(* IEC 61131-3 sources: automatic-screwdriver-line/src/POU/Job_Handler, 6 files *)

(* ---- ErrorCodeToString.st ---- *)
// Generated from Automatic_ScrewDriver_Line.xml by tools/export_st.py - do not edit.
// The CODESYS project is the source of truth.

FUNCTION ErrorCodeToString : STRING
VAR_INPUT
	Code : ErrorCode;
END_VAR

CASE Code OF
	ErrorCode.NoError :
		ErrorCodeToString := 'No Error';
	ErrorCode.EnablementError:
		ErrorCodeToString := 'Enablement Error';
	ErrorCode.ScrewNotReleased:
		ErrorCodeToString := 'Screw Not Released';
	ErrorCode.TargetNotReached:
		ErrorCodeToString := 'Target Not Reached';
	ErrorCode.SpindleError:
		ErrorCodeToString := 'Spindle Error';
	ErrorCode.CobotNotConnected:
		ErrorCodeToString := 'Cobot Not Connected';
	ErrorCode.CobotMovementNotReached:
		ErrorCodeToString := 'Cobot Movement Not Reached';
	ErrorCode.RtcNotAvailable:
		ErrorCodeToString := 'Rtc Not Available';
ELSE
		ErrorCodeToString := 'Unknown Error';
END_CASE

END_FUNCTION

(* ---- Trace.st ---- *)
// Generated from Automatic_ScrewDriver_Line.xml by tools/export_st.py - do not edit.
// The CODESYS project is the source of truth.

FUNCTION Trace : BOOL
VAR_INPUT
	Severity : UDINT;   // LogClass.LOG_INFO / LOG_WARNING / LOG_ERROR
	Msg : STRING(255);
END_VAR

LogAdd(
	hLogger   := CmpLog.LogConstants.LOG_STD_LOGGER,
	stCmpName := Machine_Constants.LOG_COMPONENT_NAME,
	diClassID := UDINT_TO_DINT(Severity),
	diErrorID := 0,
	diInfoID  := 0,
	stInfo    := Msg
);

Trace := TRUE;

END_FUNCTION

(* ---- FB_JobManager.st ---- *)
// Generated from Automatic_ScrewDriver_Line.xml by tools/export_st.py - do not edit.
// The CODESYS project is the source of truth.

FUNCTION_BLOCK FB_JobManager EXTENDS FB_FunctionBlock_Base
VAR
	_InitDone : BOOL;
	_state : JobState;
	_ActiveError : ErrorCode;
	_Stop : BOOL;
	_Reseters : ARRAY[1..6] OF I_Resettable;
	_Diagnosable : ARRAY[1..6] OF I_Diagnosable;
	_i : DINT;
	_UserInterface : REFERENCE TO FB_UserInterface;
	_JobSelector : REFERENCE TO FB_JobSelector;
	_Mover : I_Mover;
	_zAxis : REFERENCE TO FB_zAxis;
	_Spindle : REFERENCE TO FB_Spindle;
	_ReportJob : REFERENCE TO FB_ReportJob;
	_SpindleOk : BOOL;
	_MoverOk : BOOL;
END_VAR

METHOD Reset : BOOL

ClearError();
Reset := TRUE;
END_METHOD

METHOD Init : BOOL
VAR_INPUT
	UserInterface : REFERENCE TO FB_UserInterface;
	JobSelector : REFERENCE TO FB_JobSelector;
	Mover : I_Mover;
	zAxis : REFERENCE TO FB_zAxis;
	Spindle : REFERENCE TO FB_Spindle;
	ReportJob : REFERENCE TO FB_ReportJob;
END_VAR

_UserInterface REF= UserInterface;
_JobSelector REF= JobSelector;
_Mover := Mover;
_zAxis REF= zAxis;
_Spindle REF= Spindle;
_ReportJob REF= ReportJob;

// Reseters
_Reseters[1] := _UserInterface;
_Reseters[2] := _JobSelector;
_Reseters[3] := _Mover;
_Reseters[4] := _zAxis;
_Reseters[5] := _Spindle;
_Reseters[6] := _ReportJob;

// Diagnosable
_Diagnosable[1] := _UserInterface;
_Diagnosable[2] := _JobSelector;
_Diagnosable[3] := _Mover;
_Diagnosable[4] := _zAxis;
_Diagnosable[5] := _Spindle;
_Diagnosable[6] := _ReportJob;

_InitDone := TRUE;
Init := TRUE;
END_METHOD

METHOD DisableAll : BOOL

_SpindleOk := _Spindle.Disable();
_MoverOk   := _Mover.Disable();
DisableAll := _SpindleOk AND _MoverOk;
END_METHOD

METHOD EnableAll : BOOL

_SpindleOk := _Spindle.Enable();
_MoverOk   := _Mover.Enable();
EnableAll  := _SpindleOk AND _MoverOk;
END_METHOD

METHOD ResetAll : BOOL

ResetAll := TRUE;

FOR _i := 1 TO UPPER_BOUND(_Reseters, 1) DO
    IF NOT _Reseters[_i].Reset() THEN
        ResetAll := FALSE;
    END_IF
END_FOR
END_METHOD

METHOD CheckErrors : ErrorCode

CheckErrors := ErrorCode.NoError;

FOR _i := 1 TO UPPER_BOUND(_Diagnosable, 1) DO
    IF _Diagnosable[_i].GetError() <> ErrorCode.NoError
       AND CheckErrors = ErrorCode.NoError THEN
        CheckErrors := _Diagnosable[_i].GetError();
    END_IF
END_FOR
END_METHOD

METHOD RunJob : BOOL

IF NOT _InitDone THEN
	RETURN;
END_IF

_ActiveError := CheckErrors();
_Stop := _UserInterface.IsStopRequired();

IF _ActiveError <> ErrorCode.NoError AND _state <> JobState.Reset THEN
    _state := JobState.Error;
END_IF

IF _state <> JobState.Reset AND _state <> JobState.Error THEN
    EnableAll();
ELSE
    DisableAll();
END_IF

CASE _state OF
	JobState.Reset :
		IF ResetAll() THEN
			_state := JobState.Idle;
		END_IF
	JobState.Idle:
		IF _Stop THEN
			_state := JobState.Reset;
		ELSIF _zAxis.Retract() THEN
        	IF _UserInterface.IsStartRequired() THEN
            _ReportJob.Reset();
			_ReportJob.JobStart();
            _state := JobState.ReadingTargetPosition;
        	END_IF
    	END_IF
	JobState.ReadingTargetPosition :
		IF _JobSelector.ReturnScrew() THEN
			_state:= JobState.MovingToTargetPosition;
		ELSE
			_state := JobState.MovingToBase;
		END_IF
	JobState.MovingToTargetPosition :
		IF _Mover.MoveToPosition(_JobSelector.CurrentScrew.PositionMm) THEN
			_state:= JobState.MovingZaxisToTool;
		END_IF
	JobState.MovingZaxisToTool :
		    CASE _zAxis.Engage() OF
        		ActionResult.Done:
            		_state := JobState.ProcessingTool;
				ActionResult.Failed:
            		_ReportJob.FailScrew(_JobSelector.CurrentScrew);
					_state := JobState.MovingZaxisToBase;
    		END_CASE
	JobState.ProcessingTool :
		IF _Spindle.ProcessTool(_JobSelector.CurrentScrew.AngleDeg) THEN
			_ReportJob.SuccessScrew(_JobSelector.CurrentScrew);
			_state:= JobState.MovingZaxisToBase;
		END_IF
	JobState.MovingZaxisToBase :
		IF _zAxis.Retract() THEN
			_state:= JobState.ReadingTargetPosition;
		END_IF
	JobState.MovingToBase :
		IF _Mover.MoveToPosition(0)  THEN
			_state := JobState.Idle;
			_ReportJob.JobEnd();
		END_IF
	JobState.Error :
		IF _Stop THEN
			_state := JobState.Reset;
		END_IF
END_CASE

// Stop during a job = abort: publish the partial report, then reset every component.
// The next Start begins a fresh job from the first screw.
IF _Stop
   AND _state <> JobState.Idle
   AND _state <> JobState.Reset
   AND _state <> JobState.Error THEN
	_ReportJob.JobAborted();
	_state := JobState.Reset;
END_IF
END_METHOD

END_FUNCTION_BLOCK

(* ---- FB_JobSelector.st ---- *)
// Generated from Automatic_ScrewDriver_Line.xml by tools/export_st.py - do not edit.
// The CODESYS project is the source of truth.

FUNCTION_BLOCK FB_JobSelector EXTENDS FB_FunctionBlock_Base
VAR_INPUT
	ArrScrews : ScrewList := [
		(PositionMm := 100.0, AngleDeg := 90),
		(PositionMm := 130.0, AngleDeg := 600),
		(PositionMm := 185.0, AngleDeg := -180),
		(PositionMm := 27.0, AngleDeg := 360),
		(PositionMm := 300.0, AngleDeg := 720)
	];
END_VAR
VAR_OUTPUT
	CurrentScrew : Screw;
	Job_Done : BOOL;
END_VAR
VAR
	_TableIndex : INT := 0;
END_VAR

METHOD Reset : BOOL

ClearError();
_TableIndex := 0;
Job_Done := FALSE;

Reset := TRUE;
END_METHOD

METHOD ReturnScrew : BOOL

ReturnScrew := FALSE;

IF SelectNextScrew() THEN
	CurrentScrew := ArrScrews[_TableIndex];
	ReturnScrew := TRUE;
ELSE
	CurrentScrew.PositionMm := 0.0;
	CurrentScrew.AngleDeg := 0;
END_IF
END_METHOD

METHOD SelectNextScrew : BOOL

// Method responsible for incrementing _TableIndex
SelectNextScrew := FALSE;
Job_Done := FALSE;
IF _TableIndex < UPPER_BOUND(ArrScrews, 1) THEN
	_TableIndex := _TableIndex + 1;
	SelectNextScrew := TRUE;
ELSE
	_TableIndex := 0;
	Job_Done := TRUE;
END_IF
END_METHOD

END_FUNCTION_BLOCK

(* ---- FB_LogSink.st ---- *)
// Generated from Automatic_ScrewDriver_Line.xml by tools/export_st.py - do not edit.
// The CODESYS project is the source of truth.

FUNCTION_BLOCK FB_LogSink IMPLEMENTS I_ReportSink

METHOD PublishReport : BOOL
VAR_INPUT
	Report : JobReport;
END_VAR
VAR
	_msg : STRING(255);
END_VAR

_msg := CONCAT('Job ', UDINT_TO_STRING(Report.JobId));
_msg := CONCAT(_msg,   ' finished: ');
_msg := CONCAT(_msg,   INT_TO_STRING(Report.ScrewsOk));
_msg := CONCAT(_msg,   ' ok, ');
_msg := CONCAT(_msg,   INT_TO_STRING(Report.ScrewsFailed));
_msg := CONCAT(_msg,   ' failed');

Trace(CmpLog.LogClass.LOG_INFO, _msg);

PublishReport := TRUE;
END_METHOD

END_FUNCTION_BLOCK

(* ---- FB_ReportJob.st ---- *)
// Generated from Automatic_ScrewDriver_Line.xml by tools/export_st.py - do not edit.
// The CODESYS project is the source of truth.

FUNCTION_BLOCK FB_ReportJob EXTENDS FB_FunctionBlock_Base
VAR
	_NbSuccess : INT := 0;
	_NbFail : INT := 0;
	_FailedScrews : ScrewList;
	_SuccessfulScrews : ScrewList;
	_JobDone : BOOL;
	_JobId : UDINT;
	_StartedAt : DT;
	_FinishedAt : DT;
	_Sinks : ARRAY[1..3] OF I_ReportSink;
	_EmptyScrewList : ScrewList;
END_VAR

METHOD Reset : BOOL

ClearError();
_NbSuccess := 0;
_NbFail := 0;
_JobDone := FALSE;

_FailedScrews     := _EmptyScrewList;
_SuccessfulScrews := _EmptyScrewList;

Reset := TRUE;
END_METHOD

METHOD JobEnd : BOOL

_FinishedAt := Now();

Trace(CmpLog.LogClass.LOG_INFO, 'Job Done');

JobEnd := SendReportToSinks(Completed := TRUE);
END_METHOD

METHOD SuccessScrew : BOOL
VAR_INPUT
	SuccessfulScrew : Screw;
END_VAR

SuccessScrew := FALSE;

IF _NbSuccess < UPPER_BOUND(_SuccessfulScrews, 1) THEN
	_NbSuccess := _NbSuccess + 1;
	_SuccessfulScrews[_NbSuccess] := SuccessfulScrew;
	SuccessScrew := TRUE;
END_IF

Trace(CmpLog.LogClass.LOG_INFO,
        CONCAT('Screw successfully processed at position ', REAL_TO_STRING(SuccessfulScrew.PositionMm)));
END_METHOD

METHOD FailScrew : BOOL
VAR_INPUT
	FailedScrew : Screw;
END_VAR

FailScrew := FALSE;

IF _NbFail < UPPER_BOUND(_FailedScrews, 1) THEN
	_NbFail := _NbFail + 1;
	_FailedScrews[_NbFail] := FailedScrew;
	FailScrew := TRUE;
END_IF

Trace(CmpLog.LogClass.LOG_WARNING,
        CONCAT('Screw missed at position ', REAL_TO_STRING(FailedScrew.PositionMm)));
END_METHOD

METHOD JobStart : BOOL

_JobId      := _JobId + 1;
_StartedAt  := Now();
_FinishedAt := DT#1970-01-01-00:00:00;

Trace(CmpLog.LogClass.LOG_INFO, 'Job Started');

JobStart := TRUE;
END_METHOD

METHOD JobAborted : BOOL

_FinishedAt := Now();

Trace(CmpLog.LogClass.LOG_WARNING, 'Job Aborted');

JobAborted := SendReportToSinks(Completed := FALSE);
END_METHOD

METHOD AddSink : BOOL
VAR_INPUT
	Sink : I_ReportSink;
END_VAR
VAR
	_i : DINT;
END_VAR

AddSink := FALSE;

FOR _i := 1 TO UPPER_BOUND(_Sinks, 1) DO
	IF _Sinks[_i] = 0 THEN
		_Sinks[_i] := Sink;
		AddSink := TRUE;
		RETURN;
	END_IF
END_FOR
END_METHOD

METHOD SendReportToSinks : BOOL
VAR_INPUT
	Completed : BOOL;   // TRUE = job finished normally, FALSE = aborted by operator
END_VAR
VAR
	_report : JobReport;
	_i : DINT;
END_VAR

_report.JobId        := _JobId;
_report.StartedAt    := _StartedAt;
_report.FinishedAt   := _FinishedAt;
_report.ScrewsOk     := _NbSuccess;
_report.ScrewsFailed := _NbFail;
_report.FailedScrews := _FailedScrews;
_report.Completed := Completed;

SendReportToSinks := TRUE;

FOR _i := 1 TO UPPER_BOUND(_Sinks, 1) DO
	IF _Sinks[_i] <> 0 THEN
		IF NOT _Sinks[_i].PublishReport(_report) THEN
			SendReportToSinks := FALSE;
		END_IF
	END_IF
END_FOR
END_METHOD

METHOD Now : DT
VAR
	_sec : UDINT;
	_res : RTS_IEC_RESULT;
END_VAR

_sec := SysTimeRtcGet(_res);

IF _res = Errors.ERR_OK THEN
	Now := UDINT_TO_DT(_sec);
ELSE
	Now := DT#1970-01-01-00:00:00;
	RaiseError(ErrorCode.RtcNotAvailable);
END_IF
END_METHOD

END_FUNCTION_BLOCK
